TYPE "SpeedMotor_Ctrl"
VERSION : 0.1
// Block: SpeedMotor_Ctrl
   STRUCT
      SafeStop : Bool;
      Rst : Bool;
      Power : Bool;
      MovePlus : Bool;
      MoveMinus : Bool;
      Velocity : LReal;
      Acceleration : LReal;
      Deceleration : LReal;
   END_STRUCT;

END_TYPE
